FUNCTION Set_Int_From_Buffer : Buffer_Error
VAR_INPUT
END_VAR
VAR
END_VAR

END_FUNCTION

(* stored: Version 1.1.0.1, ProductVersion 3.1.4024.10
   POU Set_Int_From_Buffer: Id {9e5abfc6-95c6-4d79-982f-a8d891386b61}, SpecialFunc None *)
